// TIA Portal V19 export
ORGANIZATION_BLOCK "Main"   // OB1, LAD, ProgramCycle
TITLE = "Main Program Sweep (Cycle)"
{ S7_Optimized_Access := 'TRUE' }
// stored: SetENOAutomatically false
   VAR_INPUT
      Initial_Call : Bool;   // Initial call of this OB
      Remanence : Bool;   // =True, if remanent data are available
   END_VAR
   VAR_TEMP   // added for the SCL form of the ladder/FBD networks
      _w1 : Bool;
      _w2 : Bool;
      _w3 : Bool;
      _w4 : Bool;
      _w5 : Bool;
      _w6 : Bool;
      _w7 : Bool;
      _w8 : Bool;
      _w9 : Bool;
      _w10 : Bool;
      _w11 : Bool;
      _w12 : Bool;
      _w13 : Bool;
      _w14 : Bool;
   END_VAR
BEGIN

REGION Network 1
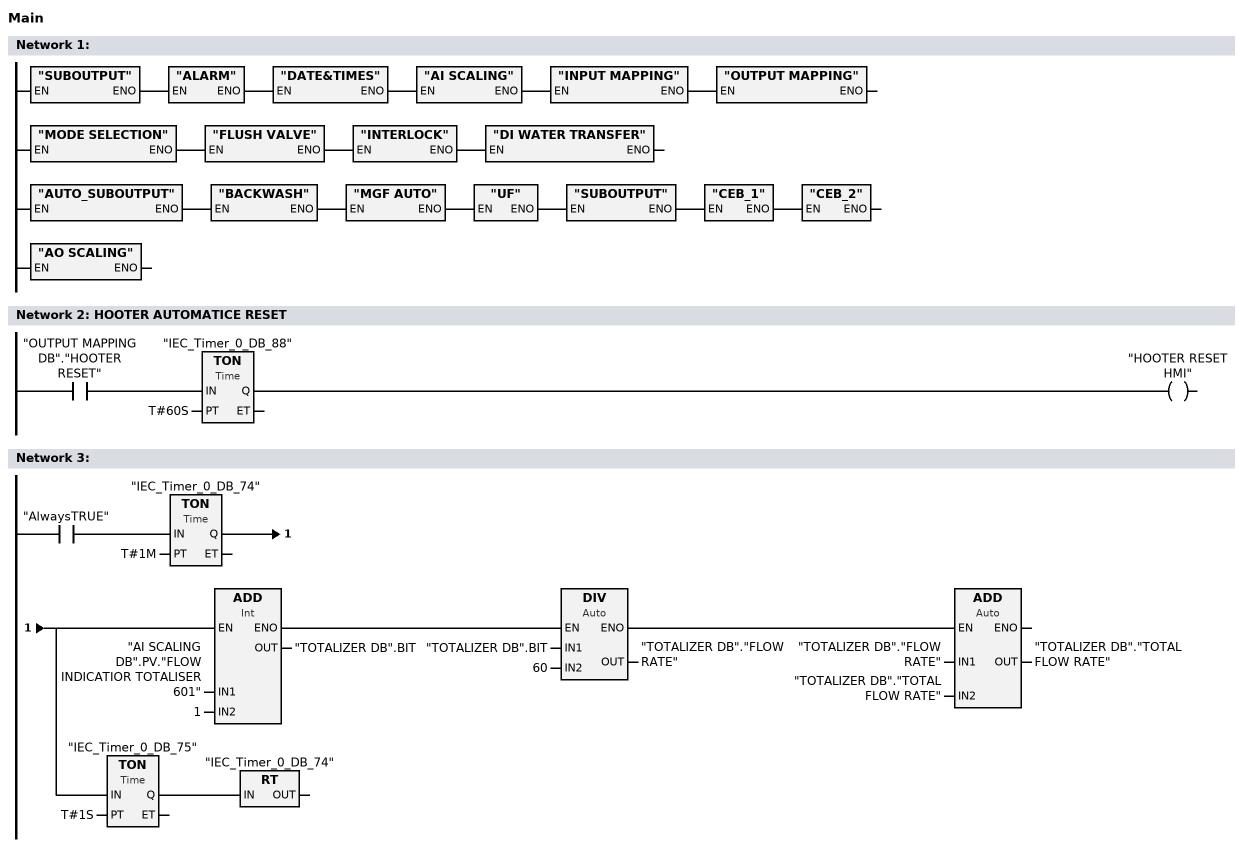
   RUNG wire#powerrail
      "SUBOUTPUT"()
      "ALARM"()
      "DATE&TIMES"()
      "AI SCALING"()
      "INPUT MAPPING"()
      "OUTPUT MAPPING"()
   END_RUNG
   RUNG wire#powerrail
      "MODE SELECTION"()
      "FLUSH VALVE"()
      "INTERLOCK"()
      "DI WATER TRANSFER"()
   END_RUNG
   RUNG wire#powerrail
      "AUTO_SUBOUTPUT"()
      "BACKWASH"()
      "MGF AUTO"()
      "UF"()
      "SUBOUTPUT"()
      "CEB_1"()
      "CEB_2"()
   END_RUNG
   RUNG wire#powerrail
      "AO SCALING"()
   END_RUNG
   // the same network as SCL:
   "SUBOUTPUT"(ENO => #_w1);
   "ALARM"(EN := #_w1, ENO => #_w2);
   "DATE&TIMES"(EN := #_w2, ENO => #_w3);
   "AI SCALING"(EN := #_w3, ENO => #_w4);
   "INPUT MAPPING"(EN := #_w4, ENO => #_w5);
   IF #_w5 THEN "OUTPUT MAPPING"(); END_IF;
   "MODE SELECTION"(ENO => #_w6);
   "FLUSH VALVE"(EN := #_w6, ENO => #_w7);
   "INTERLOCK"(EN := #_w7, ENO => #_w8);
   IF #_w8 THEN "DI WATER TRANSFER"(); END_IF;
   "AUTO_SUBOUTPUT"(ENO => #_w9);
   "BACKWASH"(EN := #_w9, ENO => #_w10);
   "MGF AUTO"(EN := #_w10, ENO => #_w11);
   "UF"(EN := #_w11, ENO => #_w12);
   "SUBOUTPUT"(EN := #_w12, ENO => #_w13);
   "CEB_1"(EN := #_w13, ENO => #_w14);
   IF #_w14 THEN "CEB_2"(); END_IF;
   "AO SCALING"();
END_REGION

REGION Network 2: HOOTER AUTOMATICE RESET
   RUNG wire#powerrail
      Contact( "OUTPUT MAPPING DB"."HOOTER RESET" )
      { S7_Templates := "time_type := Time" } "IEC_Timer_0_DB_88".TON(pt := T#60S, et =>)
      Coil( "HOOTER RESET HMI" )
   END_RUNG
   // the same network as SCL:
   "IEC_Timer_0_DB_88".TON(IN := "OUTPUT MAPPING DB"."HOOTER RESET", PT := T#60S);
   "HOOTER RESET HMI" := "IEC_Timer_0_DB_88".Q;
END_REGION

REGION Network 3
   RUNG wire#powerrail
      Contact( "AlwaysTRUE" )
      { S7_Templates := "time_type := Time" } "IEC_Timer_0_DB_74".TON(pt := T#1M, et =>)
      wire#w1
      { S7_Templates := "SrcType := Int" } Add(in1 := "AI SCALING DB".PV."FLOW INDICATIOR TOTALISER 601", in2 := 1, out => "TOTALIZER DB".BIT)
      Div(in1 := "TOTALIZER DB".BIT, in2 := 60, out => "TOTALIZER DB"."FLOW RATE")
      Add(in1 := "TOTALIZER DB"."FLOW RATE", in2 := "TOTALIZER DB"."TOTAL FLOW RATE", out => "TOTALIZER DB"."TOTAL FLOW RATE")
   END_RUNG
   RUNG wire#w1
      { S7_Templates := "time_type := Time" } "IEC_Timer_0_DB_75".TON(pt := T#1S, et =>)
      RT_Coil( "IEC_Timer_0_DB_74" )
   END_RUNG
   // the same network as SCL:
   "IEC_Timer_0_DB_74".TON(IN := "AlwaysTRUE", PT := T#1M);
   IF "IEC_Timer_0_DB_74".Q THEN
       "TOTALIZER DB".BIT := "AI SCALING DB".PV."FLOW INDICATIOR TOTALISER 601" + 1;
       "TOTALIZER DB"."FLOW RATE" := "TOTALIZER DB".BIT / 60;
       "TOTALIZER DB"."TOTAL FLOW RATE" := "TOTALIZER DB"."FLOW RATE" + "TOTALIZER DB"."TOTAL FLOW RATE";
   END_IF;
   "IEC_Timer_0_DB_75".TON(IN := "IEC_Timer_0_DB_74".Q, PT := T#1S);
   IF "IEC_Timer_0_DB_75".Q THEN RESET_TIMER("IEC_Timer_0_DB_74"); END_IF;
END_REGION
END_ORGANIZATION_BLOCK
